INTERFACE PUBLIC IdleCommands EXTENDS RunningStateCommands

METHOD PUBLIC Start
END_METHOD

END_INTERFACE

(* stored: Version 1.1.0.1, ProductVersion 3.1.4026.18
   Itf IdleCommands: Id {98a18d41-1301-03fd-1f24-fccf520ed562}
   Method Start: Id {10ff5ee6-413f-0d0d-317f-29627efddc1f} *)
